Staubli VAL3: readDetectValue.pgx

public program readDetectValue(num& x_nDetectValue[], FlagStatus& x_fSensorStatus)
  local num l_nRevData[27]
  local num l_nNumRev
  local num l_nNumTemp[27]
  local num l_nNum
  local num l_n
begin

  //This program is used for reading the detected force/torque values from the Wacoh sensor and
  //convert them to the interaction force/torque for the robot operation tasks.


  //Send the uppercase command R for inquiring the detected fore/torque values
  sClientSensor="R"
  clearBuffer(sClientSensor)
  l_nNumRev=sioGet(sClientSensor,l_nRevData)
  //Check the detected data complete or not and
  if l_nNumRev==27
    x_fSensorStatus.ForceFlag=1
  else
    x_fSensorStatus.ForceFlag=-1
    putln("Receive detected data failed!")
  endIf

  //Parse the received detected data form the Wacoh sensor
  for l_nNum=0 to 5
    //Convert the ASCII code to number
    for l_n=1 to 4
      call ASCIItoNum(l_nRevData[l_nNum*4+l_n],l_nNumTemp[l_nNum*4+l_n])
    endFor
    //Convert the detected number values to force/torque data
    x_nDetectValue[l_nNum]=l_nNumTemp[l_nNum*4+4]*1+l_nNumTemp[l_nNum*4+3]*16+l_nNumTemp[l_nNum*4+2]*256+l_nNumTemp[l_nNum*4+1]*4096
  endFor

end
